TYPE SICK_Process_Data :
STRUCT
	Q	:	BOOL;
	QoR	:	BOOL;
	Emission_Color	:	BYTE;
	value : DINT;
END_STRUCT
END_TYPE

(* stored: Version 1.1.0.1, ProductVersion 3.1.4024.10
   DUT SICK_Process_Data: Id {70ae03c8-5d35-4185-8d65-a8836b691ca9} *)
